// TIA Portal V16 export
FUNCTION "NoOp" : Void   // FC4, F_FBD
{ S7_Optimized_Access := 'TRUE' }
VERSION : 0.1
// stored: AutoNumber true, IsIECCheckEnabled false, UDAEnableTagReadback false
   VAR_IN_OUT
      "a" : Bool;
   END_VAR
BEGIN
END_FUNCTION
